// SIMATIC S7-200 project (STEP 7-Micro/WIN), CPU 224 CN REL 02.01

SYMBOL_TABLE 用户定义1
dai_hong         Q3.4     // 带(红)
dai_huang        Q3.5     // 带(黄)
dai_lan          Q3.6     // 带(兰)
kuan_hong        Q3.1     // 宽(红)
kuan_huang       Q3.2     // 宽(黄)
kuan_lan         Q3.3     // 宽(兰)
pu_hong          Q2.0     // 普(红)
pu_huang         Q2.1     // 普(黄)
pu_lan           Q2.2     // 普(兰)
yang_hong        Q2.3     // 阳(红)
yang_huang       Q2.4     // 阳(黄)
yang_lan         Q2.5     // 阳(兰)
zhong_hong       Q2.6     // 中(红)
zhong_huang      Q2.7     // 中(黄)
zhong_lan        Q3.0     // 中(兰)
END_SYMBOL_TABLE

ORGANIZATION_BLOCK 主程序:OB1
TITLE=代码包含动画管理和时钟控制模块，为2010年春节霓虹灯实现了动态灯光变换效果。 
// 当主计数器在1到8之间时，如果效果启用标志为真，系统执行“黄全亮兰中间往两边”效果：所有字的黄灯同时点亮，形成统一的黄色背景，随后兰灯从中间的中字兰灯开始，逐步向两边的阳字兰灯、宽字兰灯、普字兰灯、带字兰灯亮起，呈现流畅的动态过渡。
// 接着，当主计数器进入9到16时，若效果启用标志为真，系统切换到“红全亮兰边往中间”效果：所有字的红灯同时点亮，展现鲜艳的红色基调，同时兰灯从两端的普字兰灯和带字兰灯向中间的中字兰灯逐步亮起，带来对称的视觉冲击。
// 在17到21的范围内，系统执行“黄全亮红兰”效果，所有字的黄灯全亮，部分红灯和兰灯根据计数值逐步点亮，增添层次感。
// 随后，主计数器在22到27时触发“黄红兰交替”效果，所有字的黄灯、红灯和兰灯按时间段交替闪烁，例如22到23时亮普字黄灯等，24到25时亮普字红灯等，26到27时亮普字兰灯等，形成活泼的节奏感。
// 紧接着在28到33时，系统执行“红兰黄交替”效果，红灯、兰灯、黄灯依次点亮，保持变换的连贯性。
// 最后，当主计数器在34到43时，所有字的黄灯全亮作为背景，其他红灯和兰灯按正反顺序亮灭，例如35到36时亮普字红灯和带字兰灯，39到40时亮宽字红灯和阳字兰灯，呈现动态的追逐效果。
BEGIN
Network 1
// 网络注释
LD     SM0.5
LDW=   C11, +44
OW>=   C11, +44
O      M0.6
CTU    C11, +0
Network 2
LDW>   C11, +0
AW<=   C11, +8
A      M22.2
CALL   黄全亮（兰中间往两边）:SBR0
Network 3
LDW>=  C11, +9
AW<=   C11, +16
A      M22.2
CALL   红全亮（兰边往中间）:SBR1
Network 4
LDW>=  C11, +17
AW<=   C11, +21
CALL   黄全亮（红兰）:SBR2
Network 5
LDW>=  C11, +22
AW<=   C11, +27
CALL   黄红兰交替:SBR3
Network 6
LDW>=  C11, +28
AW<=   C11, +33
CALL   红兰黄交替:SBR4
Network 7
LDW>=  C11, +34
AW<=   C11, +43
CALL   黄全亮其余正反亮灭:SBR5
Network 8
LD     SM0.5
=      Q1.1
Network 9
LDN    SM0.5
=      Q0.6
Network 10
LDW>=  C12, +1
AW<=   C12, +2
LDW>=  C12, +3
AW<=   C12, +4
OLD
LDW>=  C12, +5
AW<=   C12, +6
OLD
LDW>=  C12, +7
AW<=   C12, +8
OLD
LDW>=  C12, +9
AW<=   C12, +10
OLD
LDW>=  C12, +11
AW<=   C12, +12
OLD
ANDW   2#1, MW10
Network 11
LDN    SM0.5
LDW>=  C12, +13
CTU    C12, +0
Network 12 // 网络标题
// 网络注释
END_ORGANIZATION_BLOCK

SUBROUTINE_BLOCK 黄全亮（兰中间往两边）:SBR0
TITLE=程序注释
BEGIN
Network 1
LDW>   C11, +1
AW<=   C11, +8
=      pu_huang:Q2.1
=      yang_huang:Q2.4
=      zhong_huang:Q2.7
=      kuan_huang:Q3.2
=      dai_huang:Q3.5
Network 2
LDW>=  C11, +2
AW<=   C11, +7
=      zhong_lan:Q3.0
Network 3
LDW>=  C11, +3
AW<=   C11, +6
=      yang_lan:Q2.5
=      kuan_lan:Q3.3
Network 4
LDW>=  C11, +4
AW<=   C11, +5
=      pu_lan:Q2.2
=      dai_lan:Q3.6
Network 17 // 网络标题
// 网络注释
Network 27 // 网络标题
// 网络注释
END_SUBROUTINE_BLOCK

SUBROUTINE_BLOCK 红全亮（兰边往中间）:SBR1
TITLE=子程序注释
BEGIN
Network 1
LDW>   C11, +9
AW<=   C11, +16
=      pu_hong:Q2.0
=      yang_hong:Q2.3
=      zhong_hong:Q2.6
=      kuan_hong:Q3.1
=      dai_hong:Q3.4
Network 2
LDW>=  C11, +10
AW<=   C11, +13
=      pu_lan:Q2.2
=      dai_lan:Q3.6
Network 3
LDW>=  C11, +11
AW<=   C11, +14
=      yang_lan:Q2.5
=      kuan_lan:Q3.3
Network 4
LDW>=  C11, +12
AW<=   C11, +15
=      zhong_lan:Q3.0
Network 5 // 网络标题
// 网络注释
END_SUBROUTINE_BLOCK

SUBROUTINE_BLOCK 黄全亮（红兰）:SBR2
TITLE=子程序注释
BEGIN
Network 1
LDW>   C11, +17
AW<=   C11, +20
=      pu_huang:Q2.1
=      yang_huang:Q2.4
=      zhong_huang:Q2.7
=      kuan_huang:Q3.2
=      dai_huang:Q3.5
Network 2 // 网络标题
// 网络注释
LDW>   C11, +18
AW<=   C11, +21
=      zhong_lan:Q3.0
=      pu_hong:Q2.0
=      dai_hong:Q3.4
Network 3
LDW>   C11, +19
AW<=   C11, +21
=      yang_lan:Q2.5
=      kuan_lan:Q3.3
=      yang_hong:Q2.3
=      kuan_hong:Q3.1
Network 4
LDW>   C11, +20
AW<=   C11, +21
=      pu_lan:Q2.2
=      dai_lan:Q3.6
=      zhong_hong:Q2.6
END_SUBROUTINE_BLOCK

SUBROUTINE_BLOCK 黄红兰交替:SBR3
TITLE=子程序注释
BEGIN
Network 1
LDW>   C11, +22
AW<=   C11, +23
=      pu_huang:Q2.1
=      yang_huang:Q2.4
=      zhong_huang:Q2.7
=      kuan_huang:Q3.2
=      dai_huang:Q3.5
Network 2
LDW>   C11, +24
AW<=   C11, +25
=      pu_hong:Q2.0
=      yang_hong:Q2.3
=      zhong_hong:Q2.6
=      kuan_hong:Q3.1
=      dai_hong:Q3.4
Network 3
LDW>   C11, +26
AW<=   C11, +27
=      pu_lan:Q2.2
=      yang_lan:Q2.5
=      zhong_lan:Q3.0
=      kuan_lan:Q3.3
=      dai_lan:Q3.6
=      M0.0
Network 4 // 网络标题
// 网络注释
END_SUBROUTINE_BLOCK

SUBROUTINE_BLOCK 红兰黄交替:SBR4
TITLE=子程序注释
BEGIN
Network 1
LDW>   C11, +28
AW<=   C11, +29
=      pu_hong:Q2.0
=      yang_hong:Q2.3
=      zhong_hong:Q2.6
=      kuan_hong:Q3.1
=      dai_hong:Q3.4
Network 2
LDW>   C11, +30
AW<=   C11, +31
=      pu_lan:Q2.2
=      yang_lan:Q2.5
=      zhong_lan:Q3.0
=      kuan_lan:Q3.3
=      dai_lan:Q3.6
=      M0.0
Network 3
LDW>   C11, +32
AW<=   C11, +33
=      pu_huang:Q2.1
=      yang_huang:Q2.4
=      zhong_huang:Q2.7
=      kuan_huang:Q3.2
=      dai_huang:Q3.5
Network 4 // 网络标题
// 网络注释
Network 14 // 网络标题
// 网络注释
END_SUBROUTINE_BLOCK

SUBROUTINE_BLOCK 黄全亮其余正反亮灭:SBR5
TITLE=子程序注释
BEGIN
Network 1
LDW>   C11, +34
AW<=   C11, +43
=      pu_huang:Q2.1
=      yang_huang:Q2.4
=      zhong_huang:Q2.7
=      kuan_huang:Q3.2
=      dai_huang:Q3.5
Network 2 // 网络标题
// 网络注释
LDW>   C11, +35
AW<=   C11, +36
=      pu_hong:Q2.0
=      dai_lan:Q3.6
Network 3
LDW>   C11, +37
AW<=   C11, +38
=      yang_hong:Q2.3
=      kuan_lan:Q3.3
Network 4
LDW>   C11, +39
AW<=   C11, +40
=      kuan_hong:Q3.1
=      yang_lan:Q2.5
Network 5
LDW>   C11, +41
AW<=   C11, +42
=      dai_hong:Q3.4
=      pu_lan:Q2.2
END_SUBROUTINE_BLOCK
